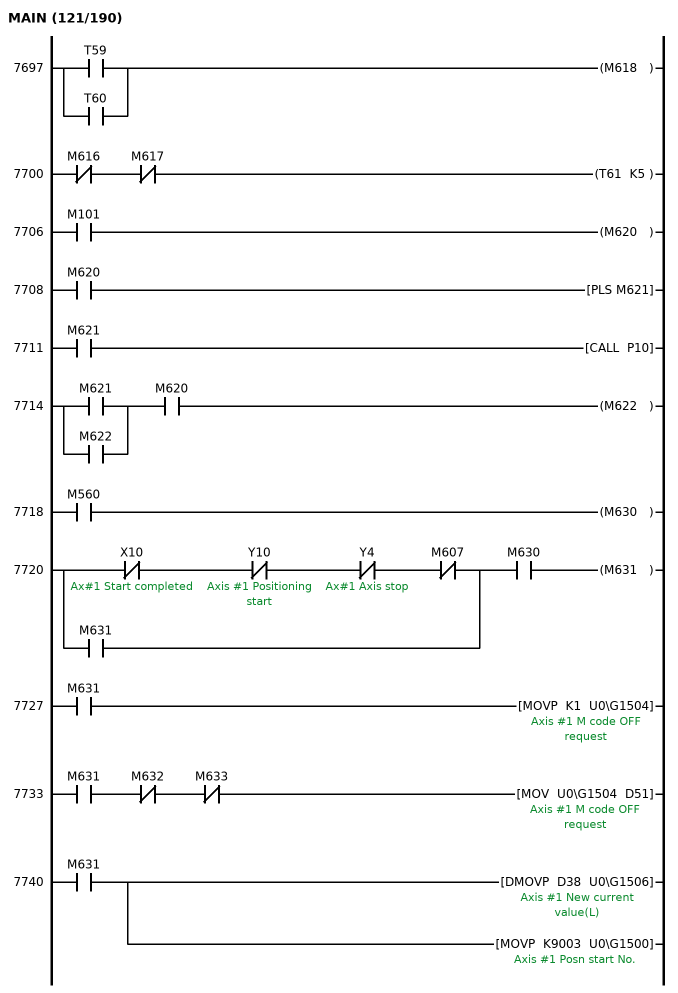
[picture p120: ladder of MAIN, rungs at steps 7697 to 7740]
7697  LD      T59
      OR      T60
      OUT     M618
7700  LDI     M616
      ANI     M617
      OUT     T61 K5
7706  LD      M101
      OUT     M620
7708  LD      M620
      PLS     M621
7711  LD      M621
      CALL    P10
7714  LD      M621
      OR      M622
      AND     M620
      OUT     M622
7718  LD      M560
      OUT     M630
7720  LDI     X10  ; Ax#1 Start completed
      ANI     Y10  ; Axis #1 Positioning start
      ANI     Y4  ; Ax#1 Axis stop
      ANI     M607
      OR      M631
      AND     M630
      OUT     M631
7727  LD      M631
      MOVP    K1 U0\G1504  ; Axis #1 M code OFF request
7733  LD      M631
      ANI     M632
      ANI     M633
      MOV     U0\G1504 D51
7740  LD      M631
      DMOVP   D38 U0\G1506  ; Axis #1 New current value(L)
      MOVP    K9003 U0\G1500
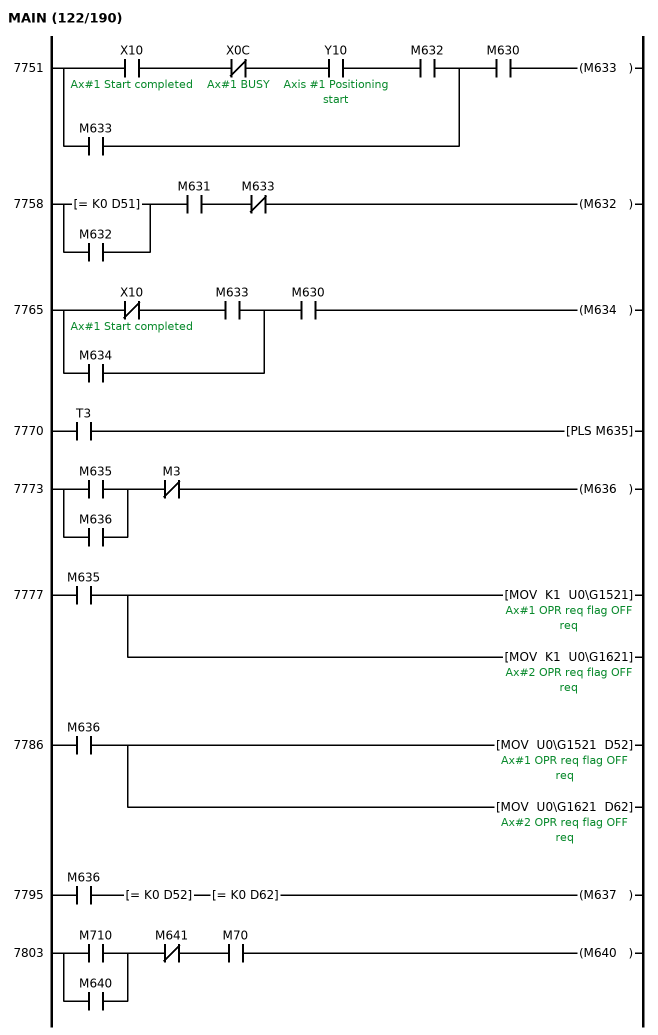
7751  LD      X10  ; Ax#1 Start completed
      ANI     X0C  ; Ax#1 BUSY
      AND     Y10  ; Axis #1 Positioning start
      AND     M632
      OR      M633
      AND     M630
      OUT     M633
7758  LD=     K0 D51
      OR      M632
      AND     M631
      ANI     M633
      OUT     M632
7765  LDI     X10  ; Ax#1 Start completed
      AND     M633
      OR      M634
      AND     M630
      OUT     M634
7770  LD      T3
      PLS     M635
7773  LD      M635
      OR      M636
      ANI     M3
      OUT     M636
7777  LD      M635
      MOV     K1 U0\G1521  ; Ax#1 OPR req flag OFF req
      MOV     K1 U0\G1621  ; Ax#2 OPR req flag OFF req
7786  LD      M636
      MOV     U0\G1521 D52
      MOV     U0\G1621 D62
7795  LD      M636
      AND=    K0 D52
      AND=    K0 D62
      OUT     M637
7803  LD      M710
      OR      M640
      ANI     M641
      AND     M70
      OUT     M640
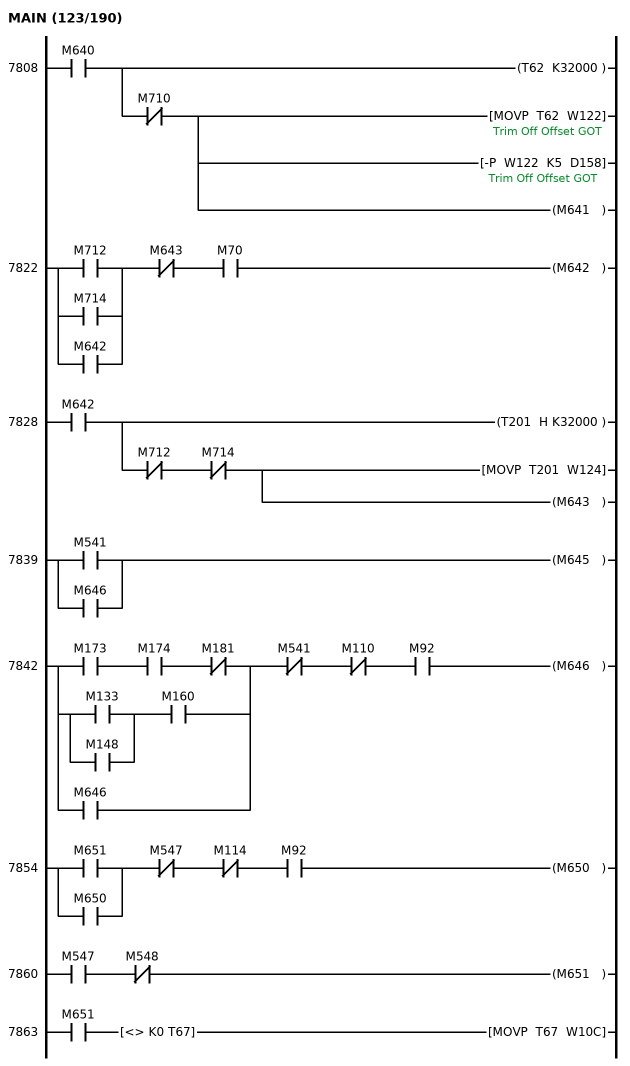
7808  LD      M640
      OUT     T62 K32000
      ANI     M710
      MOVP    T62 W122  ; Trim Off Offset GOT
      -P      W122 K5 D158
      OUT     M641
7822  LD      M712
      OR      M714
      OR      M642
      ANI     M643
      AND     M70
      OUT     M642
7828  LD      M642
      OUTH    T201 K32000
      ANI     M712
      ANI     M714
      MOVP    T201 W124
      OUT     M643
7839  LD      M541
      OR      M646
      OUT     M645
7842  LD      M173
      AND     M174
      ANI     M181
      LD      M133
      OR      M148
      AND     M160
      ORB
      OR      M646
      ANI     M541
      ANI     M110
      AND     M92
      OUT     M646
7854  LD      M651
      OR      M650
      ANI     M547
      ANI     M114
      AND     M92
      OUT     M650
7860  LD      M547
      ANI     M548
      OUT     M651
7863  LD      M651
      AND<>   K0 T67
      MOVP    T67 W10C
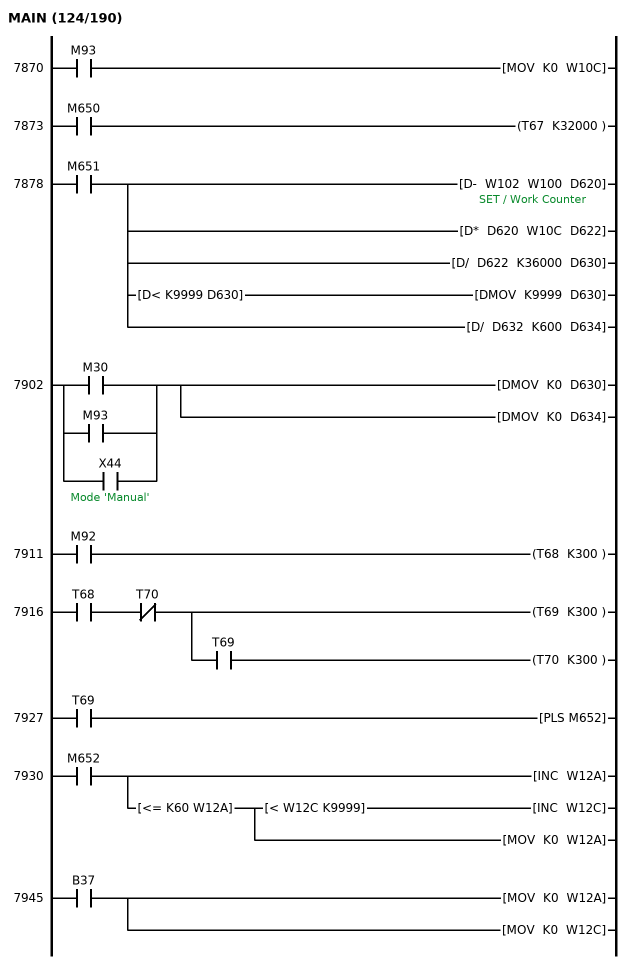
7870  LD      M93
      MOV     K0 W10C
7873  LD      M650
      OUT     T67 K32000
7878  LD      M651
      D-      W102 W100 D620
      D*      D620 W10C D622
      D/      D622 K36000 D630
      MPS
      ANDD<   K9999 D630
      DMOV    K9999 D630
      MPP
      D/      D632 K600 D634
7902  LD      M30
      OR      M93
      OR      X44  ; Mode 'Manual'
      DMOV    K0 D630
      DMOV    K0 D634
7911  LD      M92
      OUT     T68 K300
7916  LD      T68
      ANI     T70
      OUT     T69 K300
      AND     T69
      OUT     T70 K300
7927  LD      T69
      PLS     M652
7930  LD      M652
      INC     W12A
      AND<=   K60 W12A
      MPS
      AND<    W12C K9999
      INC     W12C
      MPP
      MOV     K0 W12A
7945  LD      B37
      MOV     K0 W12A
      MOV     K0 W12C
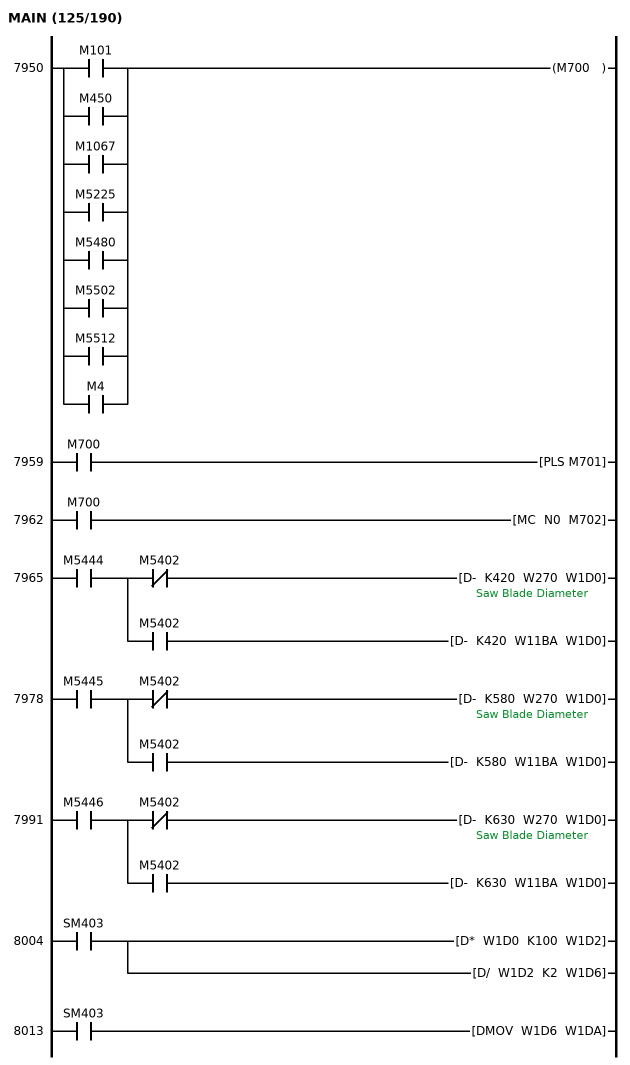
7950  LD      M101
      OR      M450
      OR      M1067
      OR      M5225
      OR      M5480
      OR      M5502
      OR      M5512
      OR      M4
      OUT     M700
7959  LD      M700
      PLS     M701
7962  LD      M700
      MC      N0 M702
7965  LD      M5444
      MPS
      ANI     M5402
      D-      K420 W270 W1D0
      MPP
      AND     M5402
      D-      K420 W11BA W1D0
7978  LD      M5445
      MPS
      ANI     M5402
      D-      K580 W270 W1D0
      MPP
      AND     M5402
      D-      K580 W11BA W1D0
7991  LD      M5446
      MPS
      ANI     M5402
      D-      K630 W270 W1D0
      MPP
      AND     M5402
      D-      K630 W11BA W1D0
8004  LD      SM403
      D*      W1D0 K100 W1D2
      D/      W1D2 K2 W1D6
8013  LD      SM403
      DMOV    W1D6 W1DA
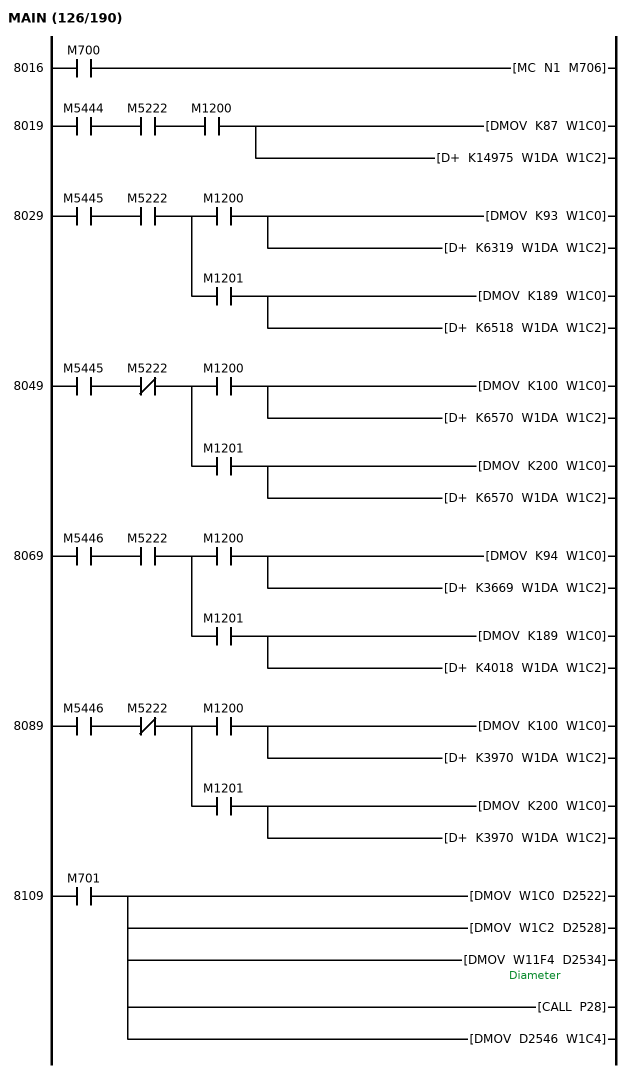
8016  LD      M700
      MC      N1 M706
8019  LD      M5444
      AND     M5222
      AND     M1200
      DMOV    K87 W1C0
      D+      K14975 W1DA W1C2
8029  LD      M5445
      AND     M5222
      MPS
      AND     M1200
      DMOV    K93 W1C0
      D+      K6319 W1DA W1C2
      MPP
      AND     M1201
      DMOV    K189 W1C0
      D+      K6518 W1DA W1C2
8049  LD      M5445
      ANI     M5222
      MPS
      AND     M1200
      DMOV    K100 W1C0
      D+      K6570 W1DA W1C2
      MPP
      AND     M1201
      DMOV    K200 W1C0
      D+      K6570 W1DA W1C2
8069  LD      M5446
      AND     M5222
      MPS
      AND     M1200
      DMOV    K94 W1C0
      D+      K3669 W1DA W1C2
      MPP
      AND     M1201
      DMOV    K189 W1C0
      D+      K4018 W1DA W1C2
8089  LD      M5446
      ANI     M5222
      MPS
      AND     M1200
      DMOV    K100 W1C0
      D+      K3970 W1DA W1C2
      MPP
      AND     M1201
      DMOV    K200 W1C0
      D+      K3970 W1DA W1C2
8109  LD      M701
      DMOV    W1C0 D2522
      DMOV    W1C2 D2528
      DMOV    W11F4 D2534
      CALL    P28
      DMOV    D2546 W1C4
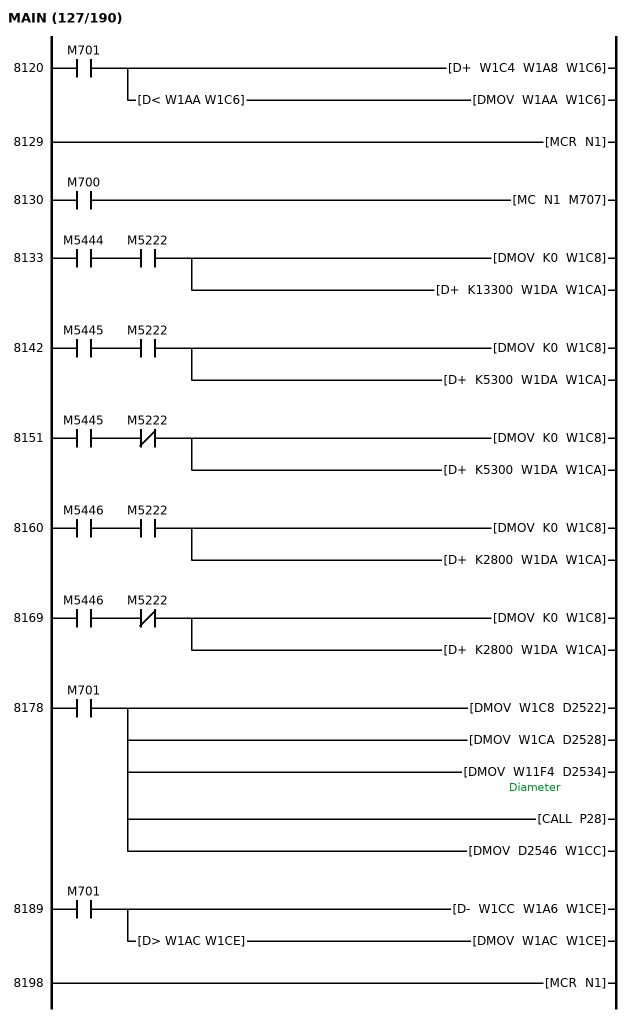
8120  LD      M701
      D+      W1C4 W1A8 W1C6
      ANDD<   W1AA W1C6
      DMOV    W1AA W1C6
8129  MCR     N1
8130  LD      M700
      MC      N1 M707
8133  LD      M5444
      AND     M5222
      DMOV    K0 W1C8
      D+      K13300 W1DA W1CA
8142  LD      M5445
      AND     M5222
      DMOV    K0 W1C8
      D+      K5300 W1DA W1CA
8151  LD      M5445
      ANI     M5222
      DMOV    K0 W1C8
      D+      K5300 W1DA W1CA
8160  LD      M5446
      AND     M5222
      DMOV    K0 W1C8
      D+      K2800 W1DA W1CA
8169  LD      M5446
      ANI     M5222
      DMOV    K0 W1C8
      D+      K2800 W1DA W1CA
8178  LD      M701
      DMOV    W1C8 D2522
      DMOV    W1CA D2528
      DMOV    W11F4 D2534
      CALL    P28
      DMOV    D2546 W1CC
8189  LD      M701
      D-      W1CC W1A6 W1CE
      ANDD>   W1AC W1CE
      DMOV    W1AC W1CE
8198  MCR     N1
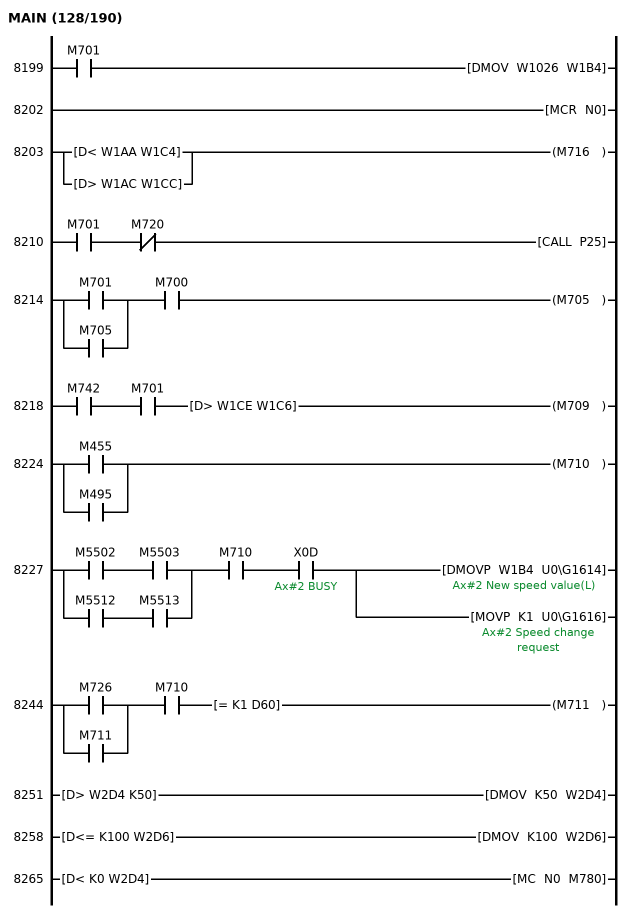
8199  LD      M701
      DMOV    W1026 W1B4
8202  MCR     N0
8203  LDD<    W1AA W1C4
      ORD>    W1AC W1CC
      OUT     M716
8210  LD      M701
      ANI     M720
      CALL    P25
8214  LD      M701
      OR      M705
      AND     M700
      OUT     M705
8218  LD      M742
      AND     M701
      ANDD>   W1CE W1C6
      OUT     M709
8224  LD      M455
      OR      M495
      OUT     M710
8227  LD      M5502
      AND     M5503
      LD      M5512
      AND     M5513
      ORB
      AND     M710
      AND     X0D  ; Ax#2 BUSY
      DMOVP   W1B4 U0\G1614  ; Ax#2 New speed value(L)
      MOVP    K1 U0\G1616  ; Ax#2 Speed change request
8244  LD      M726
      OR      M711
      AND     M710
      AND=    K1 D60
      OUT     M711
8251  LDD>    W2D4 K50
      DMOV    K50 W2D4
8258  LDD<=   K100 W2D6
      DMOV    K100 W2D6
8265  LDD<    K0 W2D4
      MC      N0 M780
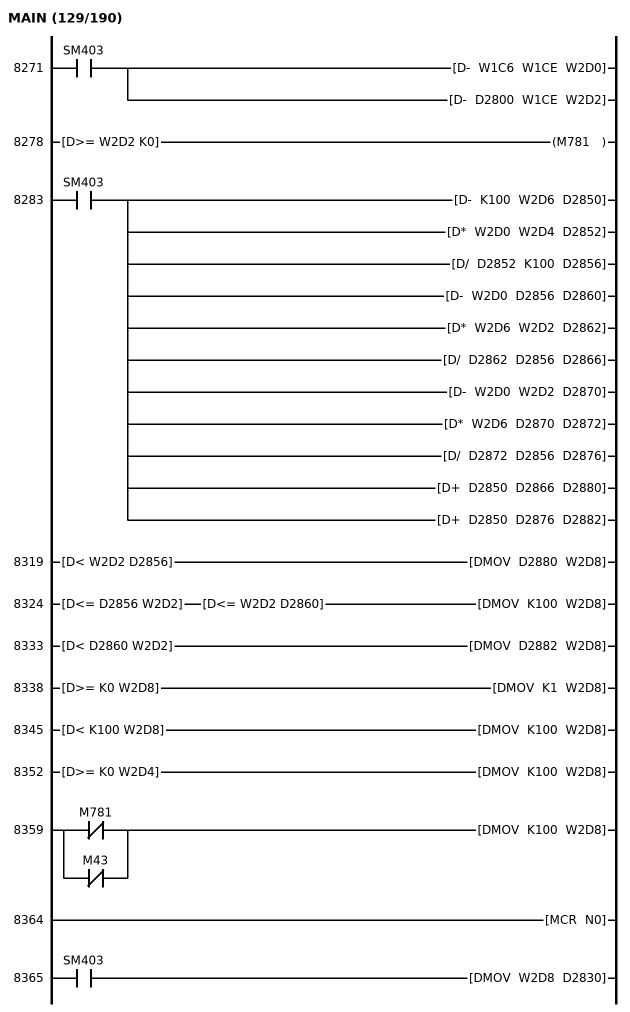
8271  LD      SM403
      D-      W1C6 W1CE W2D0
      D-      D2800 W1CE W2D2
8278  LDD>=   W2D2 K0
      OUT     M781
8283  LD      SM403
      D-      K100 W2D6 D2850
      D*      W2D0 W2D4 D2852
      D/      D2852 K100 D2856
      D-      W2D0 D2856 D2860
      D*      W2D6 W2D2 D2862
      D/      D2862 D2856 D2866
      D-      W2D0 W2D2 D2870
      D*      W2D6 D2870 D2872
      D/      D2872 D2856 D2876
      D+      D2850 D2866 D2880
      D+      D2850 D2876 D2882
8319  LDD<    W2D2 D2856
      DMOV    D2880 W2D8
8324  LDD<=   D2856 W2D2
      ANDD<=  W2D2 D2860
      DMOV    K100 W2D8
8333  LDD<    D2860 W2D2
      DMOV    D2882 W2D8
8338  LDD>=   K0 W2D8
      DMOV    K1 W2D8
8345  LDD<    K100 W2D8
      DMOV    K100 W2D8
8352  LDD>=   K0 W2D4
      DMOV    K100 W2D8
8359  LDI     M781
      ORI     M43
      DMOV    K100 W2D8
8364  MCR     N0
8365  LD      SM403
      DMOV    W2D8 D2830
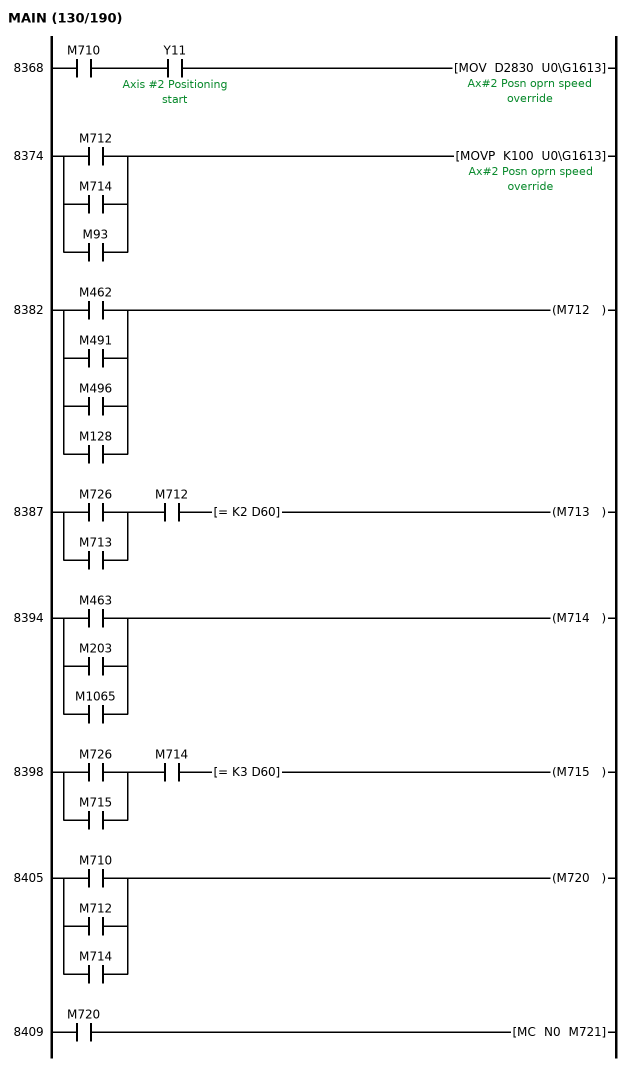
8368  LD      M710
      AND     Y11  ; Axis #2 Positioning start
      MOV     D2830 U0\G1613  ; Ax#2 Posn oprn speed override
8374  LD      M712
      OR      M714
      OR      M93
      MOVP    K100 U0\G1613
8382  LD      M462
      OR      M491
      OR      M496
      OR      M128
      OUT     M712
8387  LD      M726
      OR      M713
      AND     M712
      AND=    K2 D60
      OUT     M713
8394  LD      M463
      OR      M203
      OR      M1065
      OUT     M714
8398  LD      M726
      OR      M715
      AND     M714
      AND=    K3 D60
      OUT     M715
8405  LD      M710
      OR      M712
      OR      M714
      OUT     M720
8409  LD      M720
      MC      N0 M721
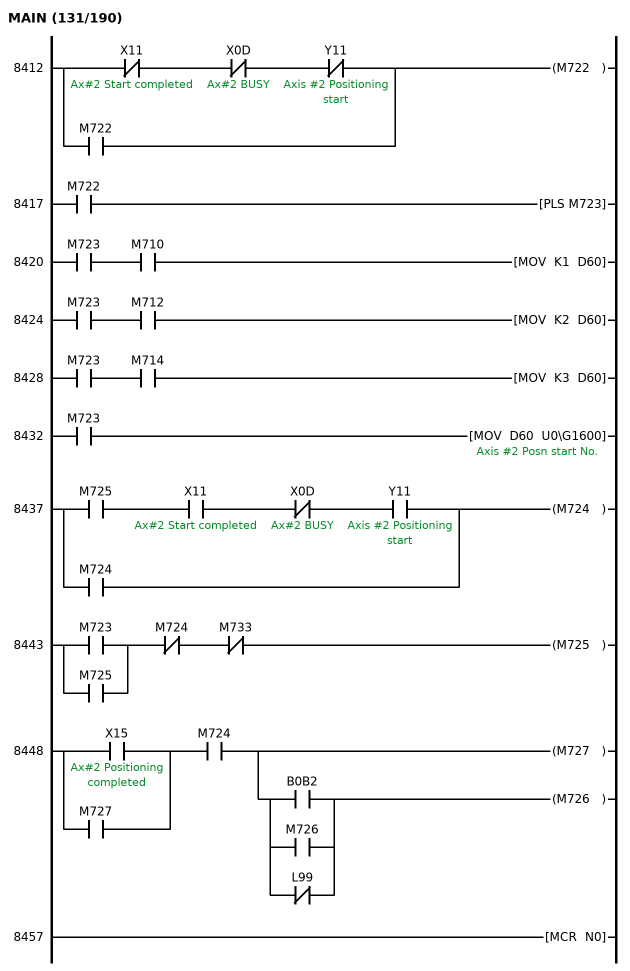
8412  LDI     X11  ; Ax#2 Start completed
      ANI     X0D  ; Ax#2 BUSY
      ANI     Y11  ; Axis #2 Positioning start
      OR      M722
      OUT     M722
8417  LD      M722
      PLS     M723
8420  LD      M723
      AND     M710
      MOV     K1 D60
8424  LD      M723
      AND     M712
      MOV     K2 D60
8428  LD      M723
      AND     M714
      MOV     K3 D60
8432  LD      M723
      MOV     D60 U0\G1600  ; Axis #2 Posn start No.
8437  LD      M725
      AND     X11  ; Ax#2 Start completed
      ANI     X0D  ; Ax#2 BUSY
      AND     Y11  ; Axis #2 Positioning start
      OR      M724
      OUT     M724
8443  LD      M723
      OR      M725
      ANI     M724
      ANI     M733
      OUT     M725
8448  LD      X15  ; Ax#2 Positioning completed
      OR      M727
      AND     M724
      OUT     M727
      LD      B0B2
      OR      M726
      ORI     L99
      ANB
      OUT     M726
8457  MCR     N0
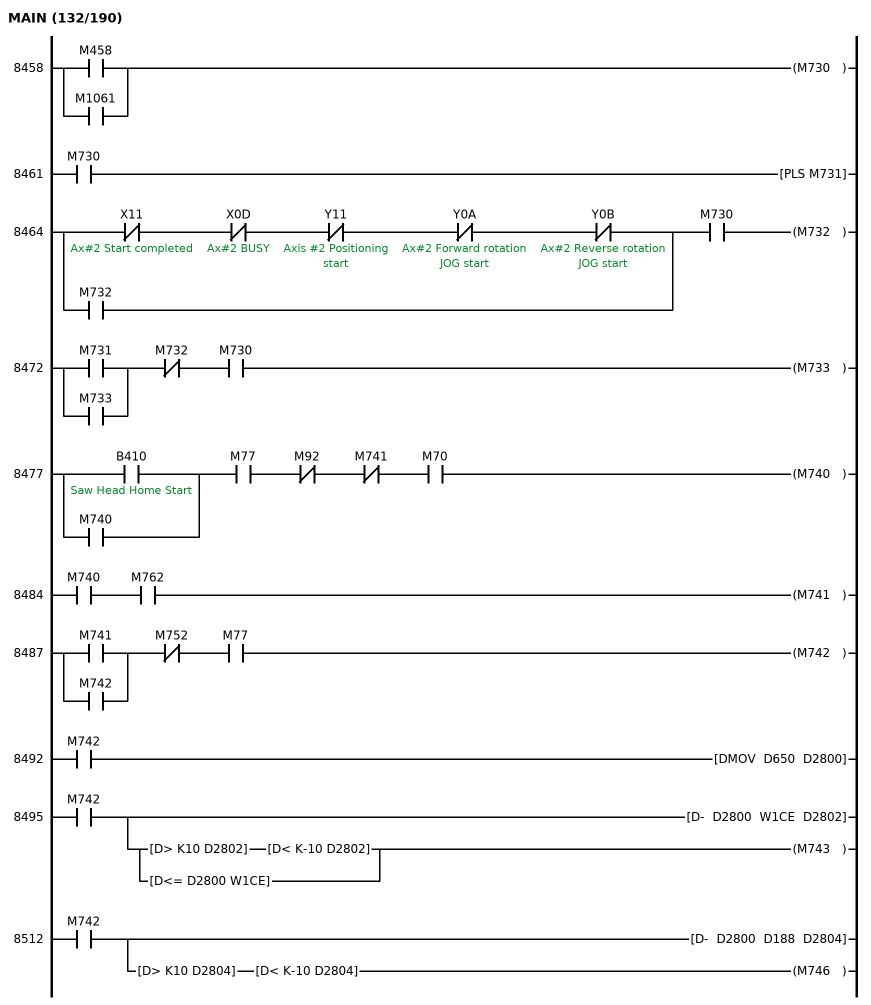
8458  LD      M458
      OR      M1061
      OUT     M730
8461  LD      M730
      PLS     M731
8464  LDI     X11  ; Ax#2 Start completed
      ANI     X0D  ; Ax#2 BUSY
      ANI     Y11  ; Axis #2 Positioning start
      ANI     Y0A  ; Ax#2 Forward rotation JOG start
      ANI     Y0B  ; Ax#2 Reverse rotation JOG start
      OR      M732
      AND     M730
      OUT     M732
8472  LD      M731
      OR      M733
      ANI     M732
      AND     M730
      OUT     M733
8477  LD      B410  ; Saw Head Home Start
      OR      M740
      AND     M77
      ANI     M92
      ANI     M741
      AND     M70
      OUT     M740
8484  LD      M740
      AND     M762
      OUT     M741
8487  LD      M741
      OR      M742
      ANI     M752
      AND     M77
      OUT     M742
8492  LD      M742
      DMOV    D650 D2800
8495  LD      M742
      D-      D2800 W1CE D2802
      LDD>    K10 D2802
      ANDD<   K-10 D2802
      ORD<=   D2800 W1CE
      ANB
      OUT     M743
8512  LD      M742
      D-      D2800 D188 D2804
      ANDD>   K10 D2804
      ANDD<   K-10 D2804
      OUT     M746
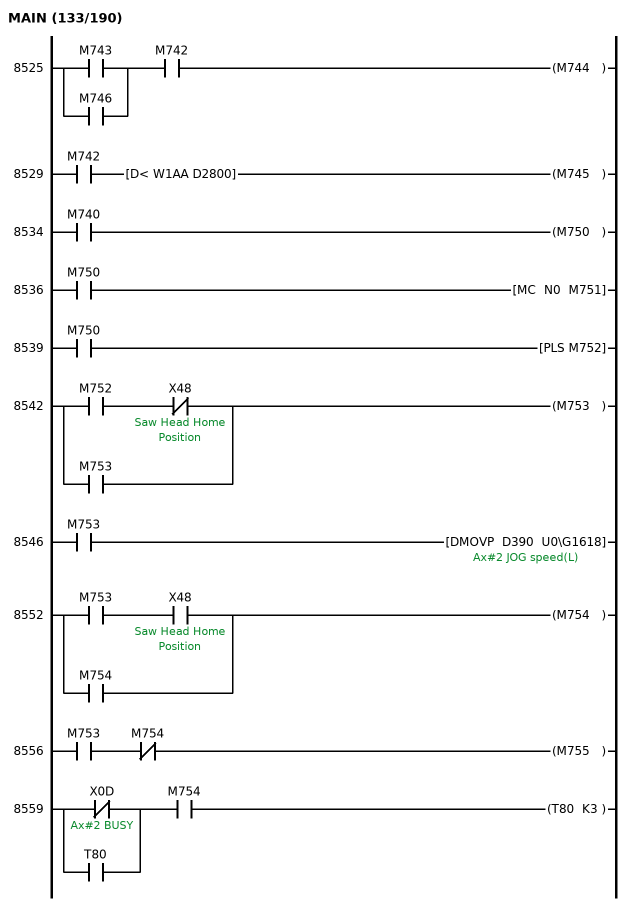
8525  LD      M743
      OR      M746
      AND     M742
      OUT     M744
8529  LD      M742
      ANDD<   W1AA D2800
      OUT     M745
8534  LD      M740
      OUT     M750
8536  LD      M750
      MC      N0 M751
8539  LD      M750
      PLS     M752
8542  LD      M752
      ANI     X48  ; Saw Head Home Position
      OR      M753
      OUT     M753
8546  LD      M753
      DMOVP   D390 U0\G1618
8552  LD      M753
      AND     X48  ; Saw Head Home Position
      OR      M754
      OUT     M754
8556  LD      M753
      ANI     M754
      OUT     M755
8559  LDI     X0D  ; Ax#2 BUSY
      OR      T80
      AND     M754
      OUT     T80 K3
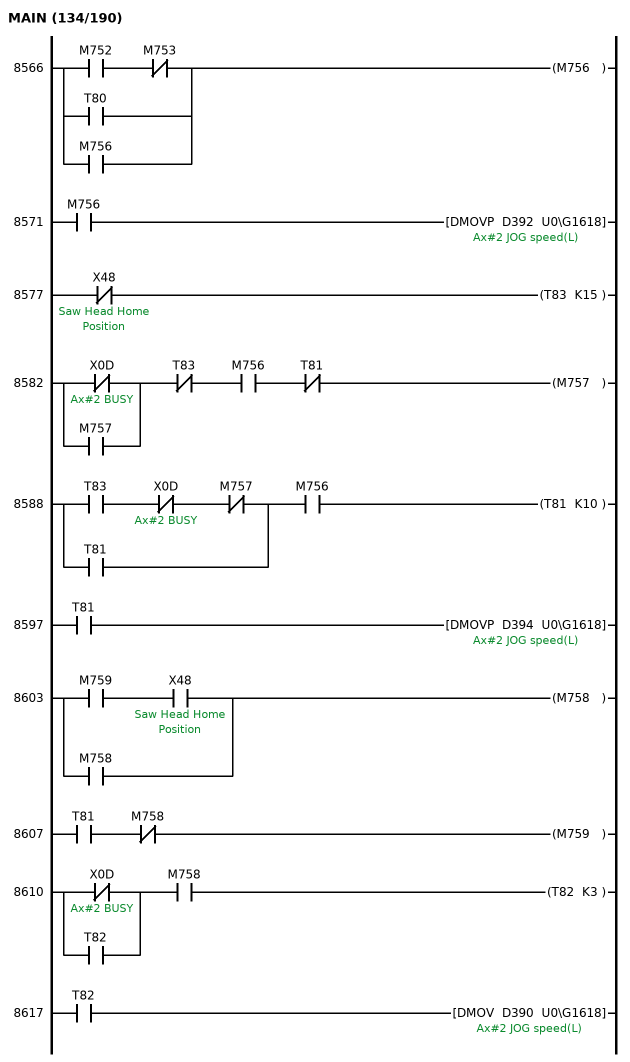
8566  LD      M752
      ANI     M753
      OR      T80
      OR      M756
      OUT     M756
8571  LD      M756
      DMOVP   D392 U0\G1618
8577  LDI     X48  ; Saw Head Home Position
      OUT     T83 K15
8582  LDI     X0D  ; Ax#2 BUSY
      OR      M757
      ANI     T83
      AND     M756
      ANI     T81
      OUT     M757
8588  LD      T83
      ANI     X0D  ; Ax#2 BUSY
      ANI     M757
      OR      T81
      AND     M756
      OUT     T81 K10
8597  LD      T81
      DMOVP   D394 U0\G1618
8603  LD      M759
      AND     X48  ; Saw Head Home Position
      OR      M758
      OUT     M758
8607  LD      T81
      ANI     M758
      OUT     M759
8610  LDI     X0D  ; Ax#2 BUSY
      OR      T82
      AND     M758
      OUT     T82 K3
8617  LD      T82
      DMOV    D390 U0\G1618
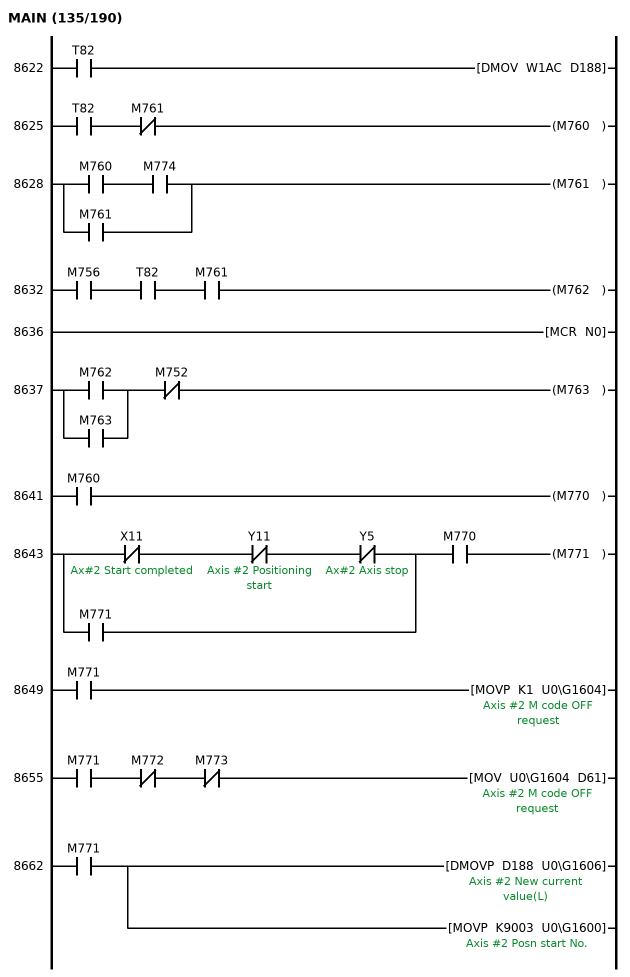
8622  LD      T82
      DMOV    W1AC D188
8625  LD      T82
      ANI     M761
      OUT     M760
8628  LD      M760
      AND     M774
      OR      M761
      OUT     M761
8632  LD      M756
      AND     T82
      AND     M761
      OUT     M762
8636  MCR     N0
8637  LD      M762
      OR      M763
      ANI     M752
      OUT     M763
8641  LD      M760
      OUT     M770
8643  LDI     X11  ; Ax#2 Start completed
      ANI     Y11  ; Axis #2 Positioning start
      ANI     Y5  ; Ax#2 Axis stop
      OR      M771
      AND     M770
      OUT     M771
8649  LD      M771
      MOVP    K1 U0\G1604  ; Axis #2 M code OFF request
8655  LD      M771
      ANI     M772
      ANI     M773
      MOV     U0\G1604 D61
8662  LD      M771
      DMOVP   D188 U0\G1606  ; Axis #2 New current value(L)
      MOVP    K9003 U0\G1600
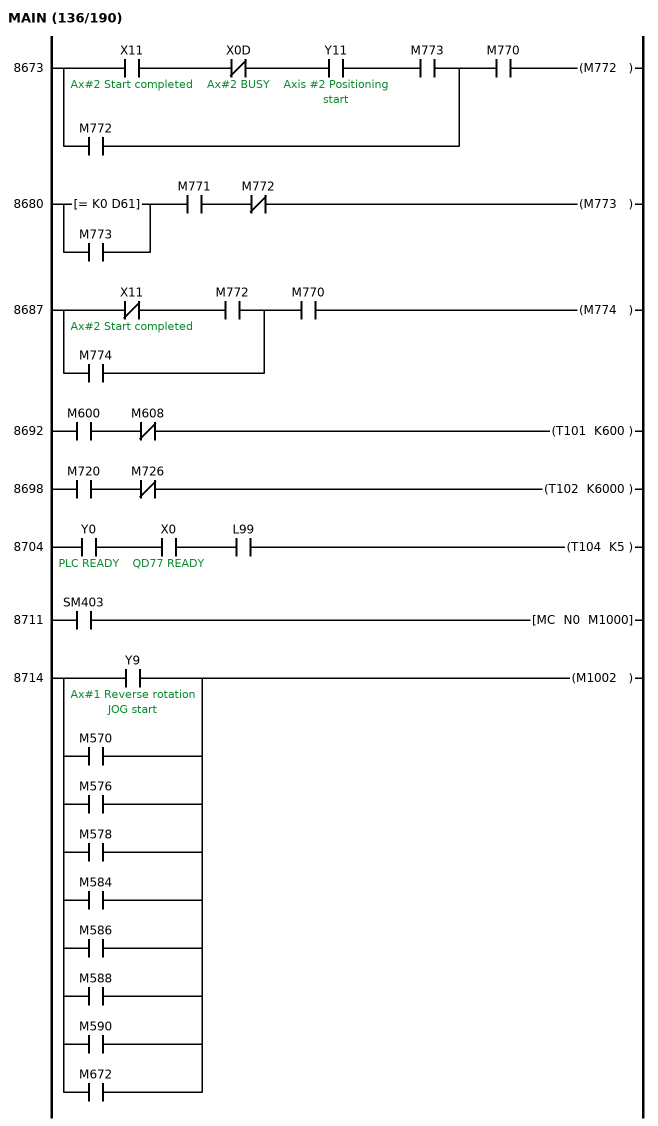
8673  LD      X11  ; Ax#2 Start completed
      ANI     X0D  ; Ax#2 BUSY
      AND     Y11  ; Axis #2 Positioning start
      AND     M773
      OR      M772
      AND     M770
      OUT     M772
8680  LD=     K0 D61
      OR      M773
      AND     M771
      ANI     M772
      OUT     M773
8687  LDI     X11  ; Ax#2 Start completed
      AND     M772
      OR      M774
      AND     M770
      OUT     M774
8692  LD      M600
      ANI     M608
      OUT     T101 K600
8698  LD      M720
      ANI     M726
      OUT     T102 K6000
8704  LD      Y0  ; PLC READY
      AND     X0  ; QD77 READY
      AND     L99
      OUT     T104 K5
8711  LD      SM403
      MC      N0 M1000
8714  LD      Y9  ; Ax#1 Reverse rotation JOG start
      OR      M570
      OR      M576
      OR      M578
      OR      M584
      OR      M586
      OR      M588
      OR      M590
      OR      M672
      OUT     M1002
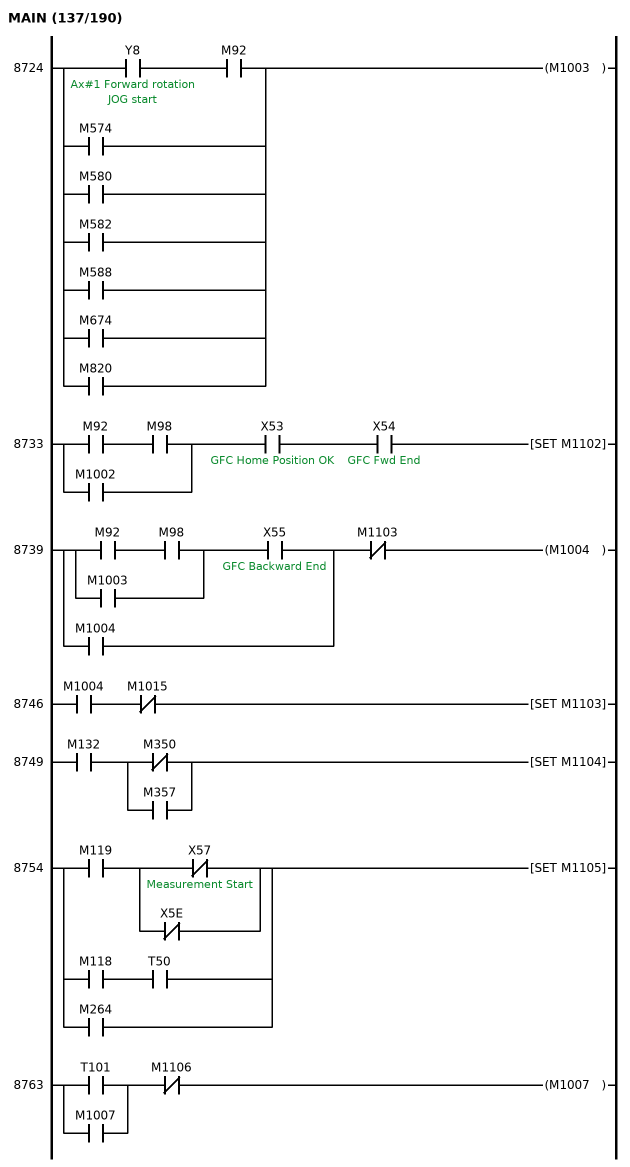
8724  LD      Y8  ; Ax#1 Forward rotation JOG start
      AND     M92
      OR      M574
      OR      M580
      OR      M582
      OR      M588
      OR      M674
      OR      M820
      OUT     M1003
8733  LD      M92
      AND     M98
      OR      M1002
      AND     X53  ; GFC Home Position OK
      AND     X54  ; GFC Fwd End
      SET     M1102
8739  LD      M92
      AND     M98
      OR      M1003
      AND     X55  ; GFC Backward End
      OR      M1004
      ANI     M1103
      OUT     M1004
8746  LD      M1004
      ANI     M1015
      SET     M1103
8749  LD      M132
      LDI     M350
      OR      M357
      ANB
      SET     M1104
8754  LD      M119
      LDI     X57  ; Measurement Start
      ORI     X5E
      ANB
      LD      M118
      AND     T50
      ORB
      OR      M264
      SET     M1105
8763  LD      T101
      OR      M1007
      ANI     M1106
      OUT     M1007
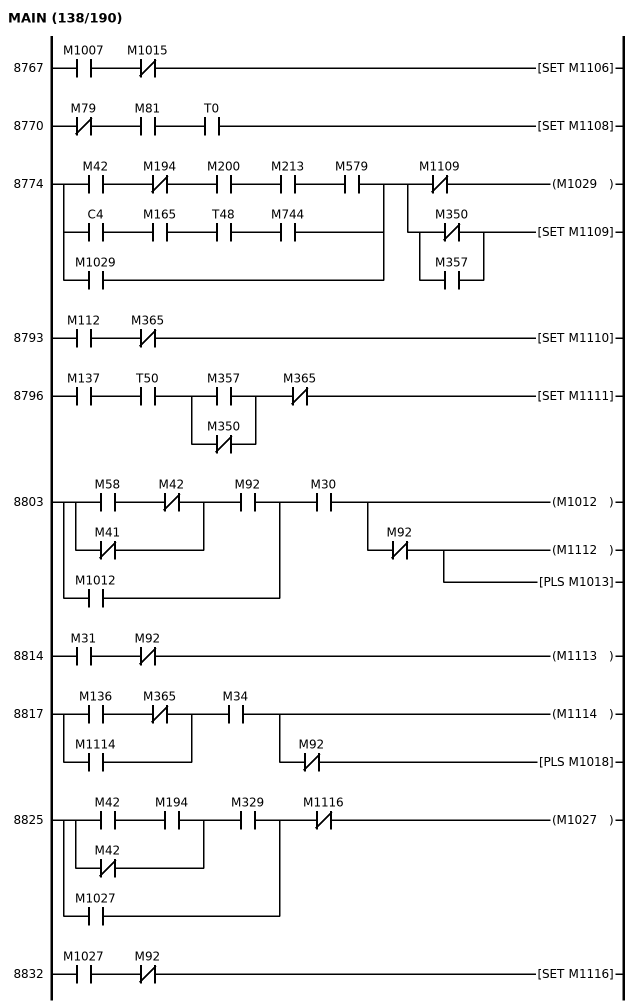
8767  LD      M1007
      ANI     M1015
      SET     M1106
8770  LDI     M79
      AND     M81
      AND     T0
      SET     M1108
8774  LD      M42
      ANI     M194
      AND     M200
      AND     M213
      AND     M579
      LD      C4
      AND     M165
      AND     T48
      AND     M744
      ORB
      OR      M1029
      MPS
      ANI     M1109
      OUT     M1029
      MPP
      LDI     M350
      OR      M357
      ANB
      SET     M1109
8793  LD      M112
      ANI     M365
      SET     M1110
8796  LD      M137
      AND     T50
      LD      M357
      ORI     M350
      ANB
      ANI     M365
      SET     M1111
8803  LD      M58
      ANI     M42
      ORI     M41
      AND     M92
      OR      M1012
      AND     M30
      OUT     M1012
      ANI     M92
      OUT     M1112
      PLS     M1013
8814  LD      M31
      ANI     M92
      OUT     M1113
8817  LD      M136
      ANI     M365
      OR      M1114
      AND     M34
      OUT     M1114
      ANI     M92
      PLS     M1018
8825  LD      M42
      AND     M194
      ORI     M42
      AND     M329
      OR      M1027
      ANI     M1116
      OUT     M1027
8832  LD      M1027
      ANI     M92
      SET     M1116
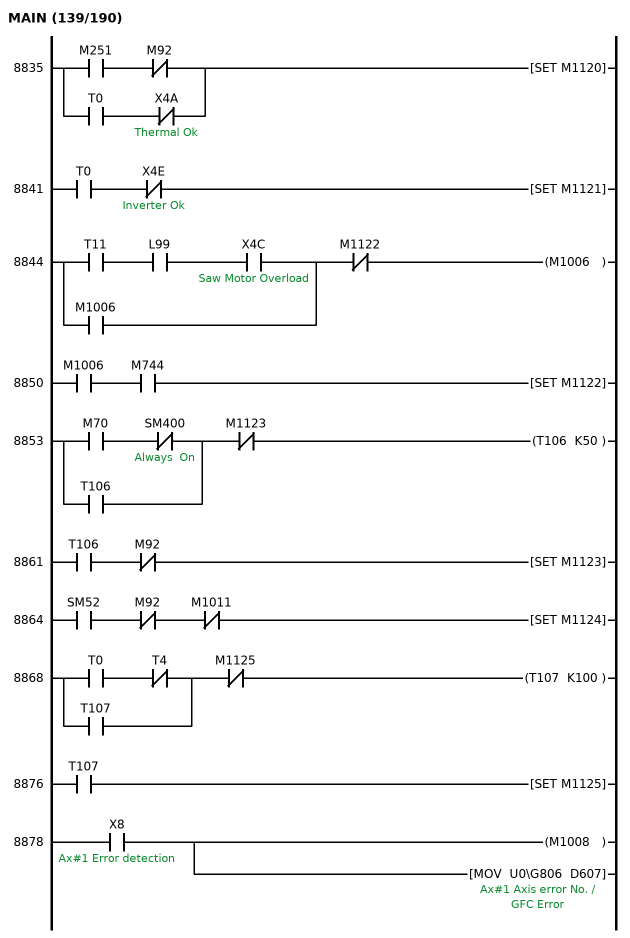
8835  LD      M251
      ANI     M92
      LD      T0
      ANI     X4A  ; Thermal Ok
      ORB
      SET     M1120
8841  LD      T0
      ANI     X4E  ; Inverter Ok
      SET     M1121
8844  LD      T11
      AND     L99
      AND     X4C  ; Saw Motor Overload
      OR      M1006
      ANI     M1122
      OUT     M1006
8850  LD      M1006
      AND     M744
      SET     M1122
8853  LD      M70
      ANI     SM400  ; Always  On
      OR      T106
      ANI     M1123
      OUT     T106 K50
8861  LD      T106
      ANI     M92
      SET     M1123
8864  LD      SM52
      ANI     M92
      ANI     M1011
      SET     M1124
8868  LD      T0
      ANI     T4
      OR      T107
      ANI     M1125
      OUT     T107 K100
8876  LD      T107
      SET     M1125
8878  LD      X8  ; Ax#1 Error detection
      OUT     M1008
      MOV     U0\G806 D607
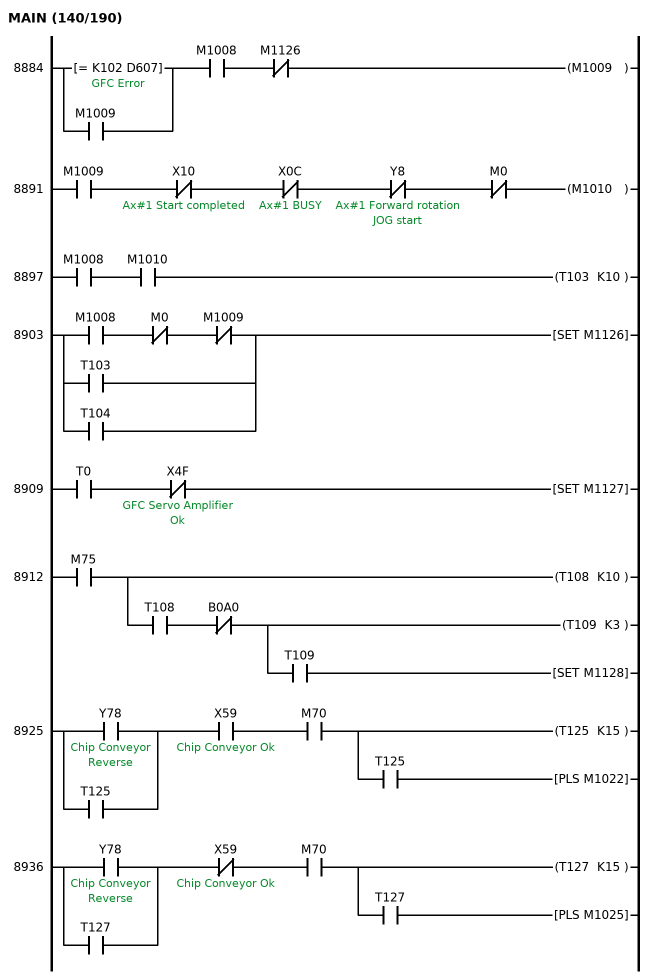
8884  LD=     K102 D607  ; GFC Error
      OR      M1009
      AND     M1008
      ANI     M1126
      OUT     M1009
8891  LD      M1009
      ANI     X10  ; Ax#1 Start completed
      ANI     X0C  ; Ax#1 BUSY
      ANI     Y8  ; Ax#1 Forward rotation JOG start
      ANI     M0
      OUT     M1010
8897  LD      M1008
      AND     M1010
      OUT     T103 K10
8903  LD      M1008
      ANI     M0
      ANI     M1009
      OR      T103
      OR      T104
      SET     M1126
8909  LD      T0
      ANI     X4F  ; GFC Servo Amplifier Ok
      SET     M1127
8912  LD      M75
      OUT     T108 K10
      AND     T108
      ANI     B0A0
      OUT     T109 K3
      AND     T109
      SET     M1128
8925  LD      Y78  ; Chip Conveyor Reverse
      OR      T125
      AND     X59  ; Chip Conveyor Ok
      AND     M70
      OUT     T125 K15
      AND     T125
      PLS     M1022
8936  LD      Y78  ; Chip Conveyor Reverse
      OR      T127
      ANI     X59  ; Chip Conveyor Ok
      AND     M70
      OUT     T127 K15
      AND     T127
      PLS     M1025
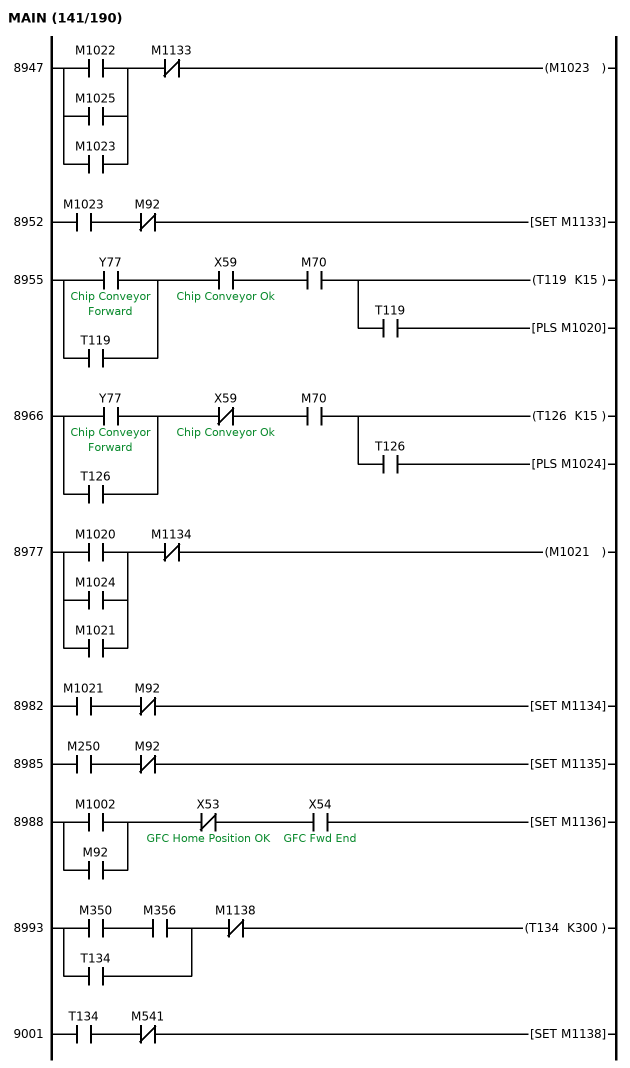
8947  LD      M1022
      OR      M1025
      OR      M1023
      ANI     M1133
      OUT     M1023
8952  LD      M1023
      ANI     M92
      SET     M1133
8955  LD      Y77  ; Chip Conveyor Forward
      OR      T119
      AND     X59  ; Chip Conveyor Ok
      AND     M70
      OUT     T119 K15
      AND     T119
      PLS     M1020
8966  LD      Y77  ; Chip Conveyor Forward
      OR      T126
      ANI     X59  ; Chip Conveyor Ok
      AND     M70
      OUT     T126 K15
      AND     T126
      PLS     M1024
8977  LD      M1020
      OR      M1024
      OR      M1021
      ANI     M1134
      OUT     M1021
8982  LD      M1021
      ANI     M92
      SET     M1134
8985  LD      M250
      ANI     M92
      SET     M1135
8988  LD      M1002
      OR      M92
      ANI     X53  ; GFC Home Position OK
      AND     X54  ; GFC Fwd End
      SET     M1136
8993  LD      M350
      AND     M356
      OR      T134
      ANI     M1138
      OUT     T134 K300
9001  LD      T134
      ANI     M541
      SET     M1138
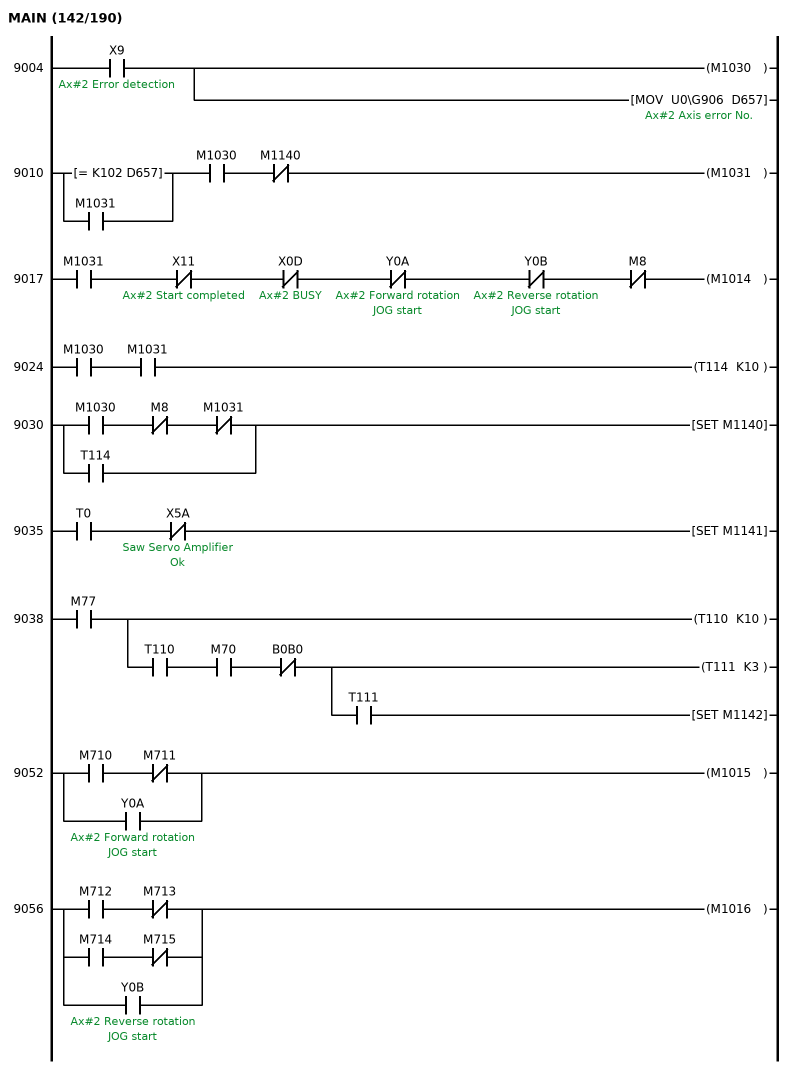
9004  LD      X9  ; Ax#2 Error detection
      OUT     M1030
      MOV     U0\G906 D657
9010  LD=     K102 D657
      OR      M1031
      AND     M1030
      ANI     M1140
      OUT     M1031
9017  LD      M1031
      ANI     X11  ; Ax#2 Start completed
      ANI     X0D  ; Ax#2 BUSY
      ANI     Y0A  ; Ax#2 Forward rotation JOG start
      ANI     Y0B  ; Ax#2 Reverse rotation JOG start
      ANI     M8
      OUT     M1014
9024  LD      M1030
      AND     M1031
      OUT     T114 K10
9030  LD      M1030
      ANI     M8
      ANI     M1031
      OR      T114
      SET     M1140
9035  LD      T0
      ANI     X5A  ; Saw Servo Amplifier Ok
      SET     M1141
9038  LD      M77
      OUT     T110 K10
      AND     T110
      AND     M70
      ANI     B0B0
      OUT     T111 K3
      AND     T111
      SET     M1142
9052  LD      M710
      ANI     M711
      OR      Y0A  ; Ax#2 Forward rotation JOG start
      OUT     M1015
9056  LD      M712
      ANI     M713
      LD      M714
      ANI     M715
      ORB
      OR      Y0B  ; Ax#2 Reverse rotation JOG start
      OUT     M1016
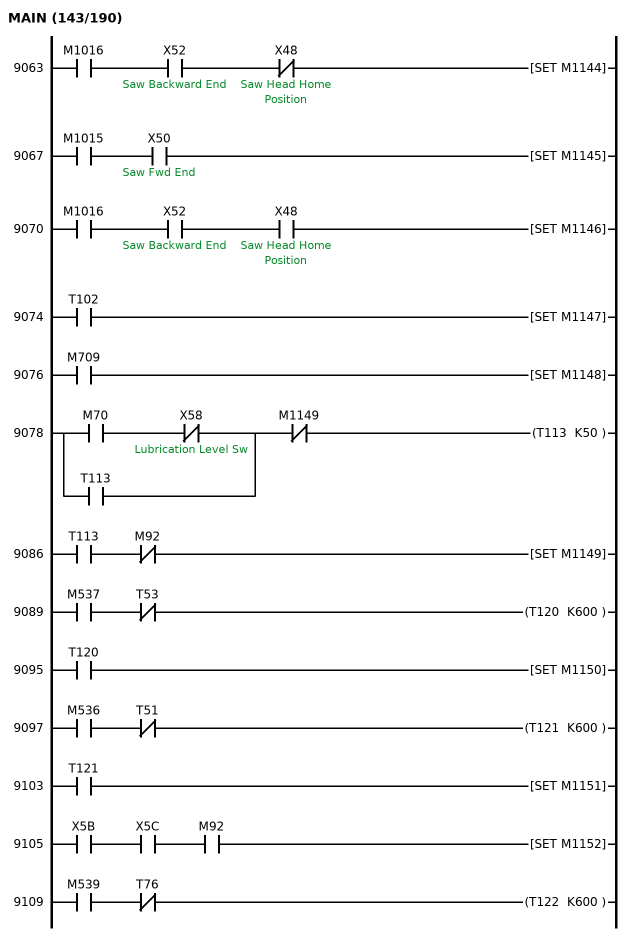
9063  LD      M1016
      AND     X52  ; Saw Backward End
      ANI     X48  ; Saw Head Home Position
      SET     M1144
9067  LD      M1015
      AND     X50  ; Saw Fwd End
      SET     M1145
9070  LD      M1016
      AND     X52  ; Saw Backward End
      AND     X48  ; Saw Head Home Position
      SET     M1146
9074  LD      T102
      SET     M1147
9076  LD      M709
      SET     M1148
9078  LD      M70
      ANI     X58  ; Lubrication Level Sw
      OR      T113
      ANI     M1149
      OUT     T113 K50
9086  LD      T113
      ANI     M92
      SET     M1149
9089  LD      M537
      ANI     T53
      OUT     T120 K600
9095  LD      T120
      SET     M1150
9097  LD      M536
      ANI     T51
      OUT     T121 K600
9103  LD      T121
      SET     M1151
9105  LD      X5B
      AND     X5C
      AND     M92
      SET     M1152
9109  LD      M539
      ANI     T76
      OUT     T122 K600
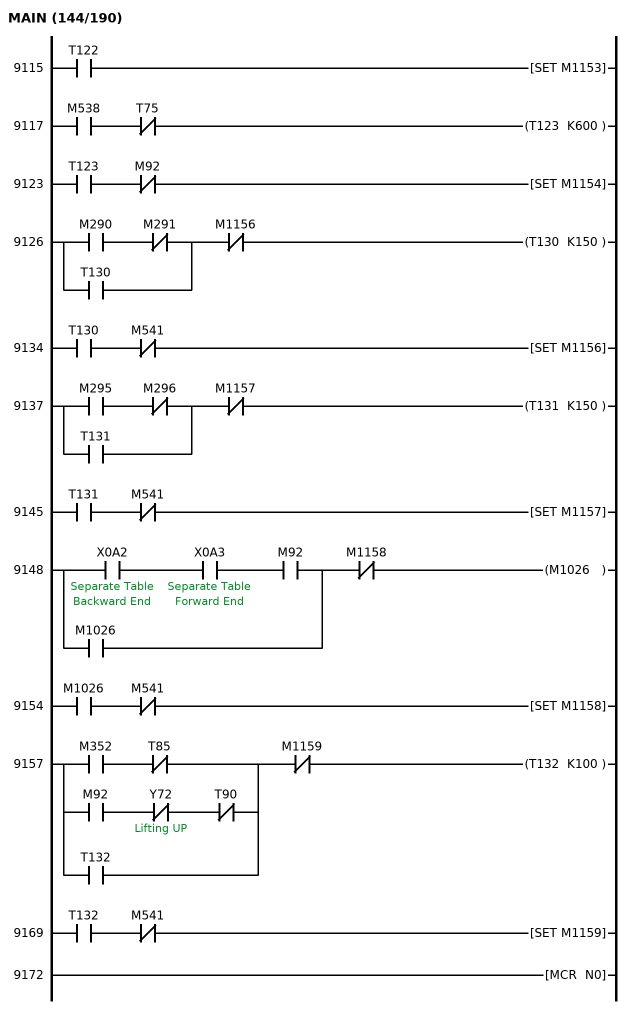
9115  LD      T122
      SET     M1153
9117  LD      M538
      ANI     T75
      OUT     T123 K600
9123  LD      T123
      ANI     M92
      SET     M1154
9126  LD      M290
      ANI     M291
      OR      T130
      ANI     M1156
      OUT     T130 K150
9134  LD      T130
      ANI     M541
      SET     M1156
9137  LD      M295
      ANI     M296
      OR      T131
      ANI     M1157
      OUT     T131 K150
9145  LD      T131
      ANI     M541
      SET     M1157
9148  LD      X0A2  ; Separate Table Backward End
      AND     X0A3  ; Separate Table Forward End
      AND     M92
      OR      M1026
      ANI     M1158
      OUT     M1026
9154  LD      M1026
      ANI     M541
      SET     M1158
9157  LD      M352
      ANI     T85
      LD      M92
      ANI     Y72  ; Lifting UP
      ANI     T90
      ORB
      OR      T132
      ANI     M1159
      OUT     T132 K100
9169  LD      T132
      ANI     M541
      SET     M1159
9172  MCR     N0
